FUNCTION_BLOCK FB_Inverter
VAR
    bEnable : BOOL;
END_VAR

END_FUNCTION_BLOCK

(* stored: POU FB_Inverter: Id {00000000-0000-0000-0000-000000000001} *)
